FUNCTION_BLOCK Sensor (* Composite Function Block Type *)
  (* Standard: 61499-2 *)
  (* Version 0.0, 5/26/2016, Andrei, nxtControl GmbH, template *)
  PACKAGE Main;
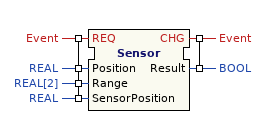
  EVENT_INPUT
    REQ WITH Position, Range, SensorPosition; (* Normal Execution Request *)
  END_EVENT
  EVENT_OUTPUT
    CHG WITH Result; (* Initialization Confirm *)
  END_EVENT
  VAR_INPUT
    Position : REAL; (* Input event qualifier *)
    Range : ARRAY [0..1] OF REAL;
    SensorPosition : REAL;
  END_VAR
  VAR_OUTPUT
    Result : BOOL; (* Output event qualifier *)
  END_VAR
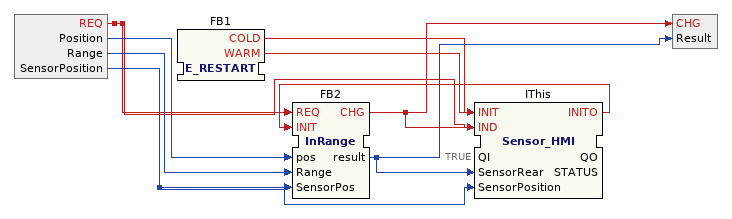
  FBS
    FB1 : E_RESTART;
    FB2 : InRange;
    IThis : Sensor_HMI(QI := TRUE);
  END_FBS
  EVENT_CONNECTIONS
    REQ TO FB2.REQ;
    FB1.COLD TO IThis.INIT;
    FB1.WARM TO IThis.INIT;
    FB2.CHG TO IThis.IND;
    IThis.INITO TO FB2.INIT;
    FB2.CHG TO CHG;
    REQ TO IThis.IND;
  END_CONNECTIONS
  DATA_CONNECTIONS
    Position TO FB2.pos;
    FB2.result TO IThis.SensorRear;
    FB2.result TO Result;
    Range TO FB2.Range;
    SensorPosition TO FB2.SensorPos;
    SensorPosition TO IThis.SensorPosition;
  END_CONNECTIONS
END_FUNCTION_BLOCK
